PROGRAM MP_4_Y103
VAR
	CompareOutput103_00: CMP_OC_DW;
	CompareOutput103_01: CMP_OC_DW;
	CompareOutput103_02: CMP_OC_DW;
	CompareOutput103_03: CMP_OC_DW;
	CompareOutput103_04: CMP_OC_DW;
	CompareOutput103_05: CMP_OC_DW;
	CompareOutput103_06: CMP_OC_DW;
	CompareOutput103_07: CMP_OC_DW;
	CompareOutput103_08: CMP_OC_DW;
	CompareOutput103_09: CMP_OC_DW;
	CompareOutput103_10: CMP_OC_DW;
	CompareOutput103_11: CMP_OC_DW;
	CompareOutput103_12: CMP_OC_DW;
	CompareOutput103_13: CMP_OC_DW;
	CompareOutput103_14: CMP_OC_DW;
	CompareOutput103_15: CMP_OC_DW;

END_VAR

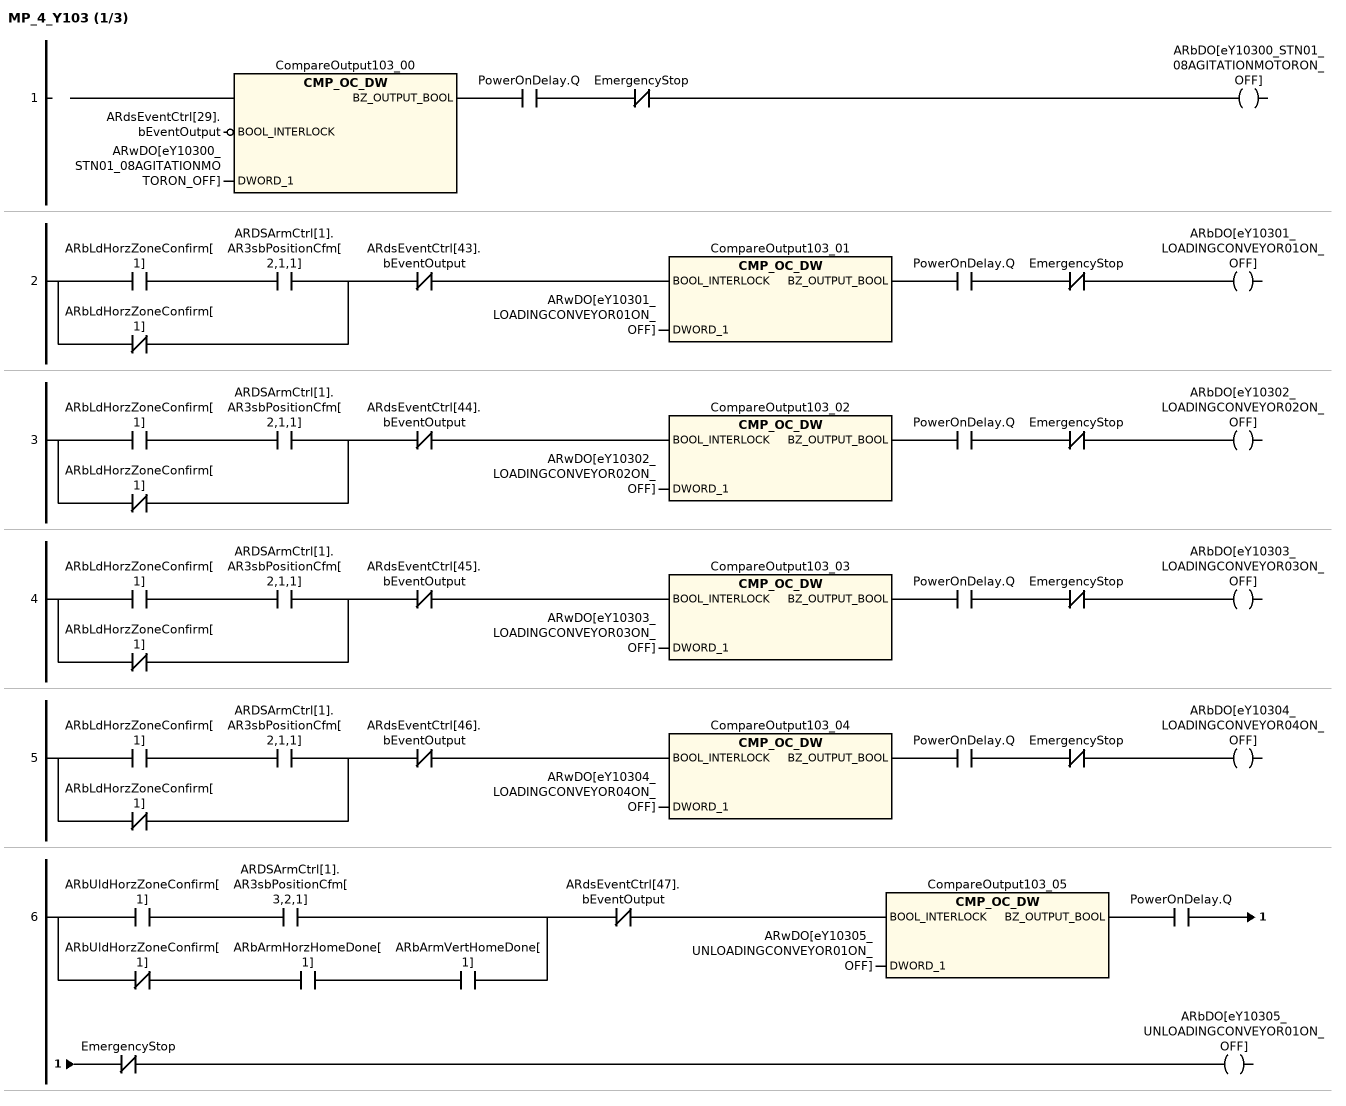
// NETWORK 1
CompareOutput103_00(BOOL_INTERLOCK := NOT ARdsEventCtrl[29].bEventOutput, DWORD_1 := ARwDO[eY10300_STN01_08AGITATIONMOTORON_OFF]); // CMP_OC_DW
ARbDO[eY10300_STN01_08AGITATIONMOTORON_OFF] := CompareOutput103_00.BZ_OUTPUT_BOOL AND PowerOnDelay.Q AND NOT EmergencyStop;

// NETWORK 2
CompareOutput103_01(BOOL_INTERLOCK := (ARbLdHorzZoneConfirm[1] AND ARDSArmCtrl[1].AR3sbPositionCfm[2,1,1] OR NOT ARbLdHorzZoneConfirm[1]) AND NOT ARdsEventCtrl[43].bEventOutput, DWORD_1 := ARwDO[eY10301_LOADINGCONVEYOR01ON_OFF]); // CMP_OC_DW
ARbDO[eY10301_LOADINGCONVEYOR01ON_OFF] := CompareOutput103_01.BZ_OUTPUT_BOOL AND PowerOnDelay.Q AND NOT EmergencyStop;

// NETWORK 3
CompareOutput103_02(BOOL_INTERLOCK := (ARbLdHorzZoneConfirm[1] AND ARDSArmCtrl[1].AR3sbPositionCfm[2,1,1] OR NOT ARbLdHorzZoneConfirm[1]) AND NOT ARdsEventCtrl[44].bEventOutput, DWORD_1 := ARwDO[eY10302_LOADINGCONVEYOR02ON_OFF]); // CMP_OC_DW
ARbDO[eY10302_LOADINGCONVEYOR02ON_OFF] := CompareOutput103_02.BZ_OUTPUT_BOOL AND PowerOnDelay.Q AND NOT EmergencyStop;

// NETWORK 4
CompareOutput103_03(BOOL_INTERLOCK := (ARbLdHorzZoneConfirm[1] AND ARDSArmCtrl[1].AR3sbPositionCfm[2,1,1] OR NOT ARbLdHorzZoneConfirm[1]) AND NOT ARdsEventCtrl[45].bEventOutput, DWORD_1 := ARwDO[eY10303_LOADINGCONVEYOR03ON_OFF]); // CMP_OC_DW
ARbDO[eY10303_LOADINGCONVEYOR03ON_OFF] := CompareOutput103_03.BZ_OUTPUT_BOOL AND PowerOnDelay.Q AND NOT EmergencyStop;

// NETWORK 5
CompareOutput103_04(BOOL_INTERLOCK := (ARbLdHorzZoneConfirm[1] AND ARDSArmCtrl[1].AR3sbPositionCfm[2,1,1] OR NOT ARbLdHorzZoneConfirm[1]) AND NOT ARdsEventCtrl[46].bEventOutput, DWORD_1 := ARwDO[eY10304_LOADINGCONVEYOR04ON_OFF]); // CMP_OC_DW
ARbDO[eY10304_LOADINGCONVEYOR04ON_OFF] := CompareOutput103_04.BZ_OUTPUT_BOOL AND PowerOnDelay.Q AND NOT EmergencyStop;

// NETWORK 6
CompareOutput103_05(BOOL_INTERLOCK := (ARbUldHorzZoneConfirm[1] AND ARDSArmCtrl[1].AR3sbPositionCfm[3,2,1] OR NOT ARbUldHorzZoneConfirm[1] AND ARbArmHorzHomeDone[1] AND ARbArmVertHomeDone[1]) AND NOT ARdsEventCtrl[47].bEventOutput, DWORD_1 := ARwDO[eY10305_UNLOADINGCONVEYOR01ON_OFF]); // CMP_OC_DW
ARbDO[eY10305_UNLOADINGCONVEYOR01ON_OFF] := CompareOutput103_05.BZ_OUTPUT_BOOL AND PowerOnDelay.Q AND NOT EmergencyStop;

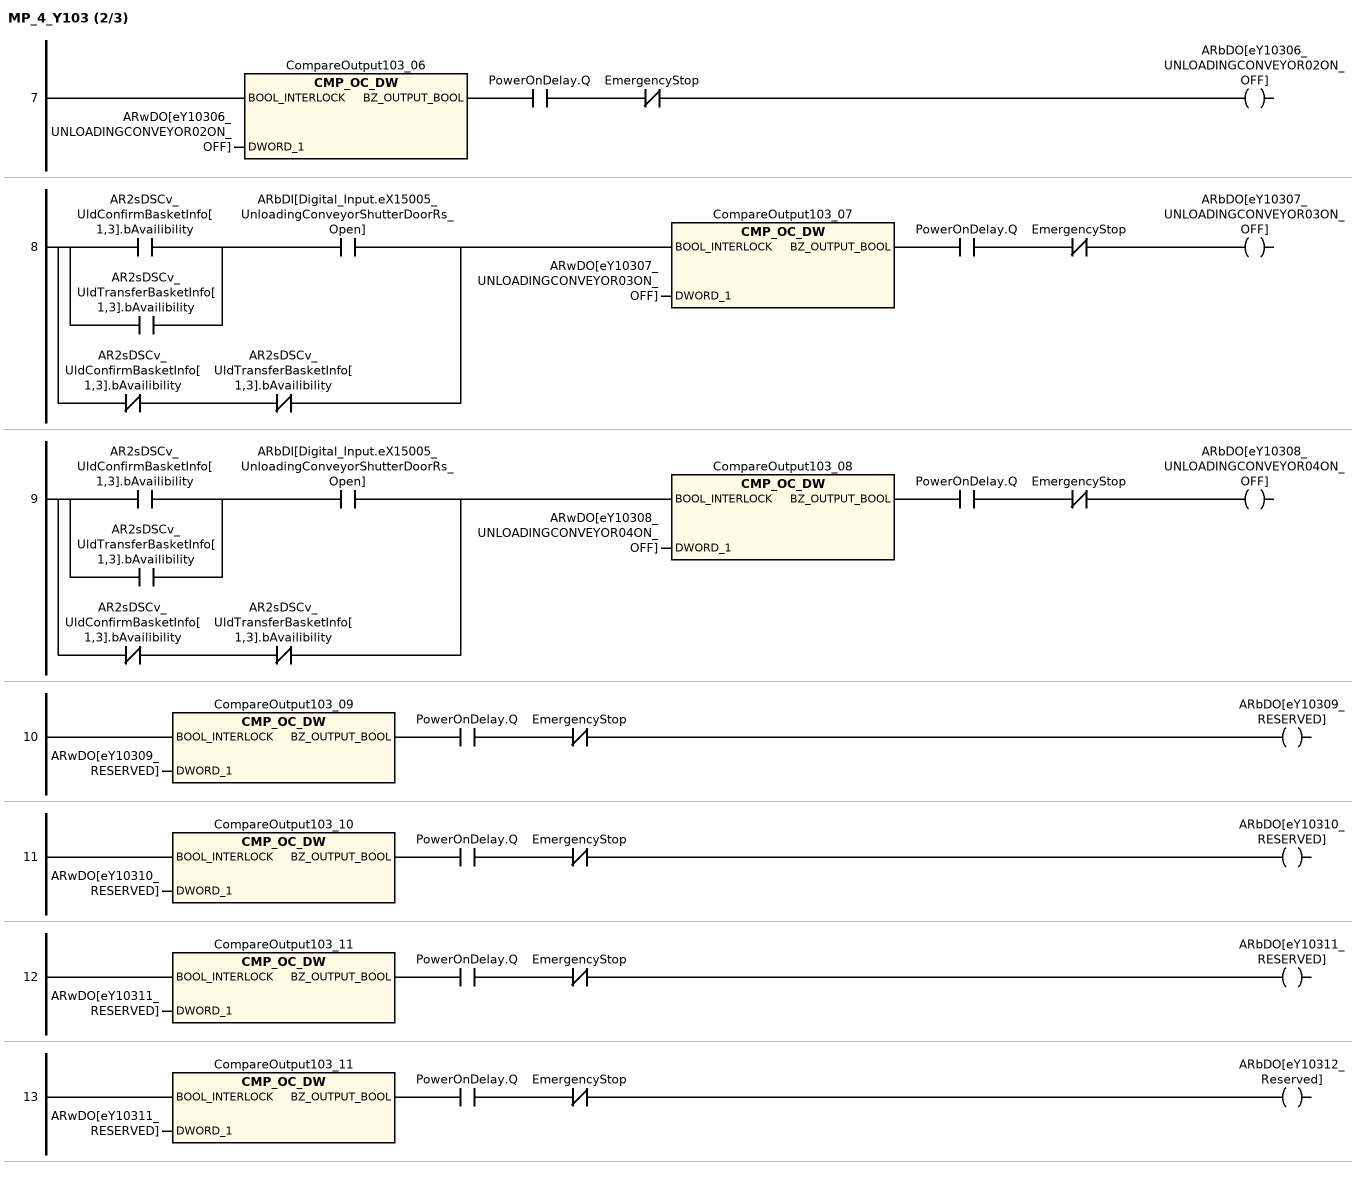
// NETWORK 7
CompareOutput103_06(BOOL_INTERLOCK := TRUE, DWORD_1 := ARwDO[eY10306_UNLOADINGCONVEYOR02ON_OFF]); // CMP_OC_DW
ARbDO[eY10306_UNLOADINGCONVEYOR02ON_OFF] := CompareOutput103_06.BZ_OUTPUT_BOOL AND PowerOnDelay.Q AND NOT EmergencyStop;

// NETWORK 8
CompareOutput103_07(BOOL_INTERLOCK := (AR2sDSCv_UldConfirmBasketInfo[1,3].bAvailibility OR AR2sDSCv_UldTransferBasketInfo[1,3].bAvailibility) AND ARbDI[Digital_Input.eX15005_UnloadingConveyorShutterDoorRs_Open] OR NOT AR2sDSCv_UldConfirmBasketInfo[1,3].bAvailibility AND NOT AR2sDSCv_UldTransferBasketInfo[1,3].bAvailibility, DWORD_1 := ARwDO[eY10307_UNLOADINGCONVEYOR03ON_OFF]); // CMP_OC_DW
ARbDO[eY10307_UNLOADINGCONVEYOR03ON_OFF] := CompareOutput103_07.BZ_OUTPUT_BOOL AND PowerOnDelay.Q AND NOT EmergencyStop;

// NETWORK 9
CompareOutput103_08(BOOL_INTERLOCK := (AR2sDSCv_UldConfirmBasketInfo[1,3].bAvailibility OR AR2sDSCv_UldTransferBasketInfo[1,3].bAvailibility) AND ARbDI[Digital_Input.eX15005_UnloadingConveyorShutterDoorRs_Open] OR NOT AR2sDSCv_UldConfirmBasketInfo[1,3].bAvailibility AND NOT AR2sDSCv_UldTransferBasketInfo[1,3].bAvailibility, DWORD_1 := ARwDO[eY10308_UNLOADINGCONVEYOR04ON_OFF]); // CMP_OC_DW
ARbDO[eY10308_UNLOADINGCONVEYOR04ON_OFF] := CompareOutput103_08.BZ_OUTPUT_BOOL AND PowerOnDelay.Q AND NOT EmergencyStop;

// NETWORK 10
CompareOutput103_09(BOOL_INTERLOCK := TRUE, DWORD_1 := ARwDO[eY10309_RESERVED]); // CMP_OC_DW
ARbDO[eY10309_RESERVED] := CompareOutput103_09.BZ_OUTPUT_BOOL AND PowerOnDelay.Q AND NOT EmergencyStop;

// NETWORK 11
CompareOutput103_10(BOOL_INTERLOCK := TRUE, DWORD_1 := ARwDO[eY10310_RESERVED]); // CMP_OC_DW
ARbDO[eY10310_RESERVED] := CompareOutput103_10.BZ_OUTPUT_BOOL AND PowerOnDelay.Q AND NOT EmergencyStop;

// NETWORK 12
CompareOutput103_11(BOOL_INTERLOCK := TRUE, DWORD_1 := ARwDO[eY10311_RESERVED]); // CMP_OC_DW
ARbDO[eY10311_RESERVED] := CompareOutput103_11.BZ_OUTPUT_BOOL AND PowerOnDelay.Q AND NOT EmergencyStop;

// NETWORK 13
CompareOutput103_11(BOOL_INTERLOCK := TRUE, DWORD_1 := ARwDO[eY10311_RESERVED]); // CMP_OC_DW
ARbDO[eY10312_Reserved] := CompareOutput103_11.BZ_OUTPUT_BOOL AND PowerOnDelay.Q AND NOT EmergencyStop;

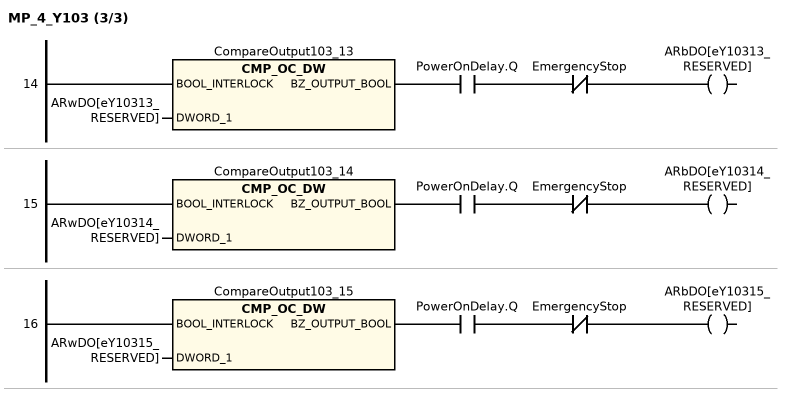
// NETWORK 14
CompareOutput103_13(BOOL_INTERLOCK := TRUE, DWORD_1 := ARwDO[eY10313_RESERVED]); // CMP_OC_DW
ARbDO[eY10313_RESERVED] := CompareOutput103_13.BZ_OUTPUT_BOOL AND PowerOnDelay.Q AND NOT EmergencyStop;

// NETWORK 15
CompareOutput103_14(BOOL_INTERLOCK := TRUE, DWORD_1 := ARwDO[eY10314_RESERVED]); // CMP_OC_DW
ARbDO[eY10314_RESERVED] := CompareOutput103_14.BZ_OUTPUT_BOOL AND PowerOnDelay.Q AND NOT EmergencyStop;

// NETWORK 16
CompareOutput103_15(BOOL_INTERLOCK := TRUE, DWORD_1 := ARwDO[eY10315_RESERVED]); // CMP_OC_DW
ARbDO[eY10315_RESERVED] := CompareOutput103_15.BZ_OUTPUT_BOOL AND PowerOnDelay.Q AND NOT EmergencyStop;

END_PROGRAM

(* stored: Version 1.1.0.1, ProductVersion 3.1.4024.11
   POU MP_4_Y103: Id {1c88166f-a5ec-4749-a2a9-d64d915f4086}, SpecialFunc None *)
